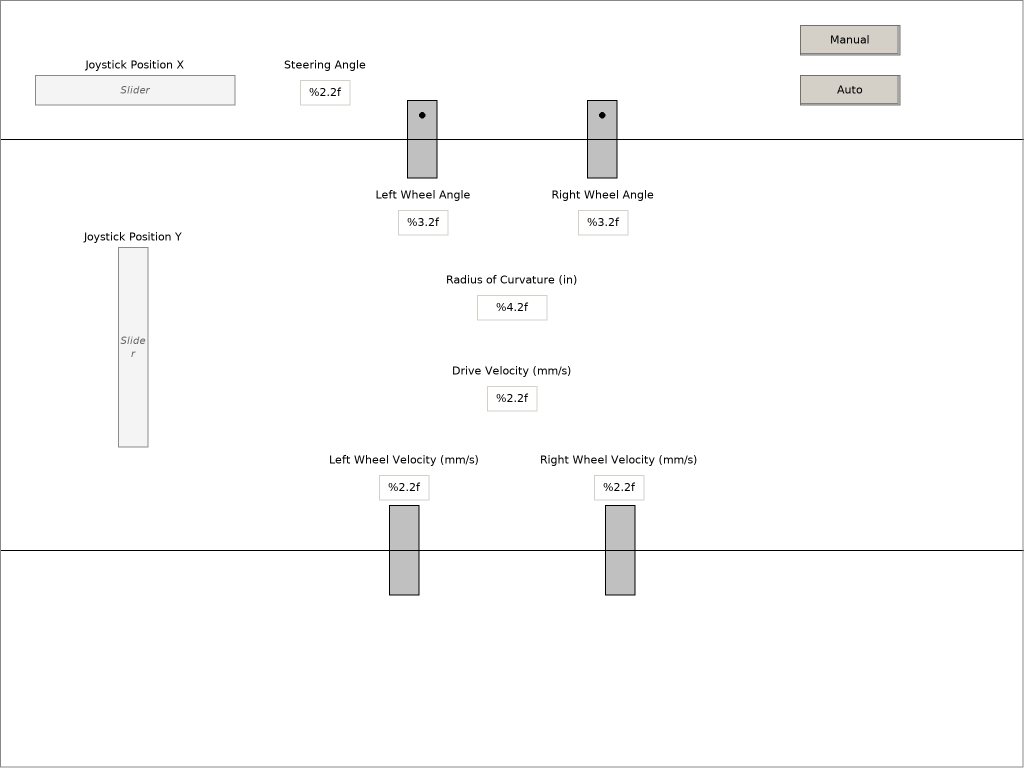
VISUALIZATION DriveSysTest  // 1024x768
    Rectangle (407,100 30x78)
        p2858320360: HARV.DriveSys.LeftWheelAngleCommand
    Rectangle (587,100 30x78)
        p2858320360: HARV.DriveSys.RightWheelAngleCommand
    Rectangle (605,505 30x90)
    Rectangle (389,505 30x90)
    Textfield (398,210 50x25), "%3.2f", text variable: HARV.DriveSys.LeftWheelAngleCommand
    Textfield (578,210 50x25), "%3.2f", text variable: HARV.DriveSys.RightWheelAngleCommand
    Textfield (379,475 50x25), "%2.2f", text variable: HARV.DriveSys.LeftVelCommand
    Textfield (594,475 50x25), "%2.2f", text variable: HARV.DriveSys.RightVelCommand
    Label (348,180 150x30), "Left Wheel Angle"
    Label (528,180 150x30), "Right Wheel Angle"
    Textfield (300,80 50x25), "%2.2f", text variable: HARV.DriveSys.SteeringAngleInput
        OnMouseClick: write the text variable via Default, min -90.0, max 90.0
    Label (250,50 150x30), "Steering Angle"
    Textfield (477,295 70x25), "%4.2f", text variable: HARV.DriveSys.ICC_R
    Label (437,265 150x30), "Radius of Curvature (in)"
    Label (324,445 160x30), "Left Wheel Velocity (mm/s)"
    Label (539,445 160x30), "Right Wheel Velocity (mm/s)"
    Textfield (487,386 50x25), "%2.2f", text variable: HARV.DriveSys.DriveVelInput
        OnMouseClick: write the text variable via Default, min -1.0, max 1.0
    Label (437,356 150x30), "Drive Velocity (mm/s)"
    Slider (35,75 200x30), variable: HARV.DriveSys.JoyStick_X, scale 0..16300
    Label (60,50 150x30), "Joystick Position X"
    Slider (118,247 30x200), variable: HARV.DriveSys.JoyStick_Y, scale 0..16300
    Label (58,222 150x30), "Joystick Position Y"
    Line (-200,139) (1224,139)
        p2858320360: HARV.DriveSys.RightWheelAngleCommand
    Line (-200,139) (1224,139)
        p2858320360: HARV.DriveSys.LeftWheelAngleCommand
    Line (0,550) (1024,550)
    Line (512,550) (512,550)
        p874137650: (HARV.DriveSys.ICC_R)*3
    Ellipse (419,112 6x6)
    Ellipse (599,112 6x6)
    Button (800,25 100x30), "Manual"
        OnMouseClick: toggle HARV.DriveSys.ManualDriveEnable
    Button (800,75 100x30), "Auto"
        OnMouseClick: toggle HARV.DriveSys.AutoDriveEnable
END_VISUALIZATION

(* stored: Version 1.1.0.1, ProductVersion 3.1.4024.12
   Visu DriveSysTest: Id {6eab1853-ea37-41ff-821c-d826b0e5034f} *)
